Staubli VAL3: diff.pgx

public program diff(num& x_nInput[], num& x_nResult[])
  local num l_nLength
  local num l_nElement
begin

  l_nLength = size(x_nInput)
  x_nResult[0] = 0
  resize(x_nResult,1,l_nLength-1)

  for l_nElement = 1 to l_nLength-1
    x_nResult[l_nElement-1] =  x_nInput[l_nElement] - x_nInput[l_nElement-1]
  endFor

end
